FUNCTION_BLOCK ECController (* Service Interface Function Block Type *)
  (* Standard: 61499-2; Description: Copyright (c) 2026 Sichuan Qunyuan Technology Co., Ltd. This program and the accompanying materials are made available under the terms of the Eclipse Public License 2.0 which is available at https://www.eclipse.org/legal/epl-2.0/ SPDX-License-Identifier: EPL-2.0 *)
  (* Version 1.0, 2026-04-09, Zijun Tang *)
  PACKAGE eclipse4diac::io::ethercat;
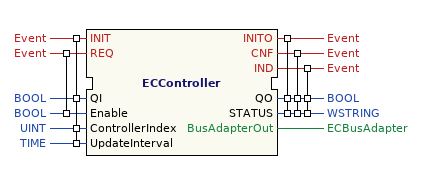
  EVENT_INPUT
    INIT WITH ControllerIndex, UpdateInterval, QI; (* Service Initialization *)
    REQ WITH Enable;
  END_EVENT
  EVENT_OUTPUT
    INITO WITH QO, STATUS; (* Initialization Confirm *)
    CNF WITH QO, STATUS; (* Confirmation of Requested Service *)
    IND WITH QO, STATUS; (* Indication from Resource *)
  END_EVENT
  VAR_INPUT
    QI : BOOL;
    Enable : BOOL;
    ControllerIndex : UINT;
    UpdateInterval : TIME := T#30us;
  END_VAR
  VAR_OUTPUT
    QO : BOOL; (* Event Output Qualifier *)
    STATUS : WSTRING; (* Service Status *)
  END_VAR
  PLUGS
    BusAdapterOut : eclipse4diac::io::ethercat::ECBusAdapter;
  END_PLUGS
END_FUNCTION_BLOCK
